// Mitsubishi GX Developer project: Station-A-GX-Mitshubishi-PLC   PLC: FX2N

PROGRAM MAIN
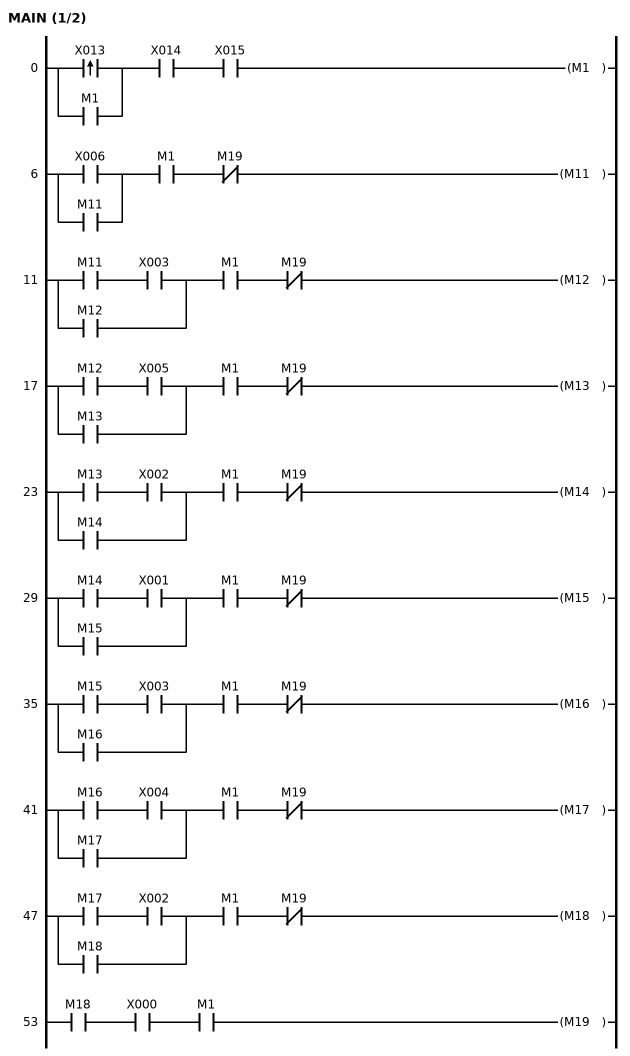
0     LDP     X013
      OR      M1
      AND     X014
      AND     X015
      OUT     M1
6     LD      X006
      OR      M11
      AND     M1
      ANI     M19
      OUT     M11
11    LD      M11
      AND     X003
      OR      M12
      AND     M1
      ANI     M19
      OUT     M12
17    LD      M12
      AND     X005
      OR      M13
      AND     M1
      ANI     M19
      OUT     M13
23    LD      M13
      AND     X002
      OR      M14
      AND     M1
      ANI     M19
      OUT     M14
29    LD      M14
      AND     X001
      OR      M15
      AND     M1
      ANI     M19
      OUT     M15
35    LD      M15
      AND     X003
      OR      M16
      AND     M1
      ANI     M19
      OUT     M16
41    LD      M16
      AND     X004
      OR      M17
      AND     M1
      ANI     M19
      OUT     M17
47    LD      M17
      AND     X002
      OR      M18
      AND     M1
      ANI     M19
      OUT     M18
53    LD      M18
      AND     X000
      AND     M1
      OUT     M19
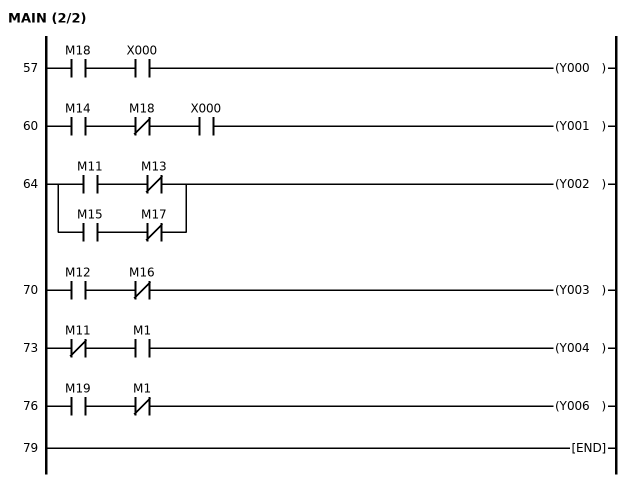
57    LD      M18
      AND     X000
      OUT     Y000
60    LD      M14
      ANI     M18
      AND     X000
      OUT     Y001
64    LD      M11
      ANI     M13
      LD      M15
      ANI     M17
      ORB
      OUT     Y002
70    LD      M12
      ANI     M16
      OUT     Y003
73    LDI     M11
      AND     M1
      OUT     Y004
76    LD      M19
      ANI     M1
      OUT     Y006
79    END
END_PROGRAM
